// TIA Portal V19 export
TYPE "Prod_Part_Target"
// stored: Access Published
   STRUCT
      Ready : Bool;   // Target pronto = Dati validi
      Tick_Mark : Bool;   // Parte deve avere Marchio identificazione spessore
      Trace_Mark : Bool;   // Parte deve avere Marchio identificazione tracciabilità
      P_ID : DInt;   // ID pezzo da assegnare
      O_ID : DInt;   // ID di produzione a cui appartiene la parte da fare
      Part_ToGo : DInt;   // Quantità parti mancanti per completare oridine.(1 = Questo è l'ultimo)
      Part_Len : Real;   // Lunghezza parte
      Part_Tol : Real;   // Tolleranza sulla lunghezza
      Beam_Code : Int;   // Codice Pezzo: 0= SG formato da una singola parte; 1= C/S = Formato da due parti accoppiate
   END_STRUCT;
END_TYPE
